Universal Robots PolyScope program: Dovetail_bottom.urp

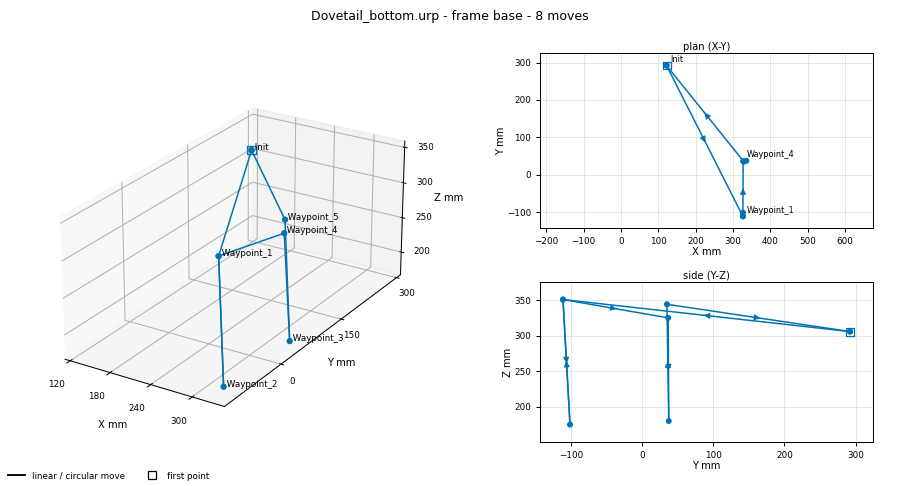
[picture p0: tool path of Dovetail_bottom.urp in frame base, 8 of 8 moves have a stored position in this frame; points joined in program order, loops and branches not executed]
Program Dovetail_bottom (installation=default directory=/programs/Mursal createdIn=5.11.11.1010533 lastSavedIn=5.11.11.1010533 robotSerialNumber=20205300864)
Calibrated DH parameters: a=[-0.000166, -0.243494, -0.153108, 0.000057, -0.000123, 0]; d=[0.151897, -1.34267, 53.988124, -52.514559, 0.085283, 0.092193]; alpha=[1.572472, -0.003756, 0.002824, 1.570807, -1.572621, 0]; deltaTheta=[0, 0.020704, 7.033215, -0.770746, 0.000004, 0]
Robot Program (runOnlyOnce=false)
  MoveL speed 250 mm/s, acceleration 1200 mm/s^2 (useActiveTCP=true) feature=Base
    Waypoint Init: TCP in base x=122.12 y=292.12 z=305.735 mm, rx=1.1346 ry=-2.9295 rz=0 rad; joints [91.64, -87.587, -91.764, -90.543, 90.034, 859.398] deg
    Waypoint Waypoint_1: TCP in base x=326.295 y=-111.364 z=350.725 mm, rx=-2.191 ry=2.2514 rz=0 rad; joints [3.411, -96.129, -70.677, -103.086, 89.973, 725.048] deg
    Waypoint Waypoint_2: TCP in base x=326.284 y=-101.463 z=174.97 mm, rx=2.191 ry=-2.2514 rz=0 rad; joints [5.115, -103.147, -111.767, -54.983, 90.02, 726.858] deg
    URCap Gripper (Robotiq_Grippers, Robotiq Inc.) dataModel(position=100.0, force=1.0, speed=0.0, positionInDouble=100.0, forceInDouble=1.0, speedInDouble=0.0, slaveIds=[9], blocking=true, robotCompliant=false)
    Waypoint Waypoint_1: TCP in base x=326.295 y=-111.364 z=350.725 mm, rx=-2.191 ry=2.2514 rz=0 rad; joints [3.411, -96.129, -70.677, -103.086, 89.973, 725.048] deg
    Waypoint Waypoint_4: TCP in base x=326.895 y=36.532 z=325.006 mm, rx=-2.1912 ry=2.2511 rz=0 rad; joints [29.747, -91.006, -83.197, -95.686, 90.011, 751.383] deg
    Waypoint Waypoint_3: TCP in base x=335.673 y=37.34 z=180.009 mm, rx=2.2548 ry=2.1875 rz=-0.0001 rad; joints [29.017, -101.53, -112.225, -56.144, 90.022, 570.937] deg
    URCap Gripper (Robotiq_Grippers, Robotiq Inc.) dataModel(position=0.0, force=1.0, speed=0.0, positionInDouble=0.0, forceInDouble=1.0, speedInDouble=0.0, slaveIds=[9], blocking=true, robotCompliant=false)
    Waypoint Waypoint_5: TCP in base x=328.908 y=34.768 z=344.077 mm, rx=-2.1932 ry=2.2493 rz=-0.0001 rad; joints [29.282, -92.138, -76.842, -100.911, 89.989, 750.812] deg
    Waypoint Init: TCP in base x=122.12 y=292.12 z=305.735 mm, rx=1.1346 ry=-2.9295 rz=0 rad; joints [91.64, -87.587, -91.764, -90.543, 90.034, 859.398] deg
